FUNCTION_BLOCK FB_SequenzReferenz IMPLEMENTS I_Sequenz
VAR_INPUT
	// Betriebsvariablen
	
	
	// Benötigter Skill
	
	// Benötigte Parameter
END_VAR
VAR_OUTPUT
END_VAR
VAR
END_VAR

METHOD M_Start : BOOL
END_METHOD

METHOD M_Stop : BOOL
END_METHOD

PROPERTY P_State : eSequenceState
GET
END_GET
END_PROPERTY

END_FUNCTION_BLOCK

(* stored: Version 1.1.0.1
   POU FB_SequenzReferenz: Id {6b767d26-9b1c-4026-9e95-eab42be9026d}, SpecialFunc None
   Method M_Start: Id {eb3028dc-dbec-4628-90f5-df6c4d441337}
   Method M_Stop: Id {7827b4f4-2c1e-4275-b842-f33cf6f9db3e}
   Property P_State: Id {7c2827b6-3c77-441b-a023-4c1a9cbde076}
   Get Get: Id {deb48184-48ba-4b82-9206-4b1433cba5a7} *)
